Staubli VAL3: stop.pgx

program stop()
begin

  //将机器人移动至总装配任务的结束点
  putln("Moving the robot to the whole assembly task end point.")
  movel(pPointRx_Asse_E,tTool_1,mMdesc_Move)
  waitEndMove()

end
